// TIA Portal V16 export
// export: Created 2022-01-12T14:34:29.2729698Z, ExportSetting WithDefaults, DisplayName Totally Integrated Automation Portal, DisplayVersion V16 Update 4, DisplayName TIA Portal Version Control Interface, DisplayVersion V16 Update 2, DisplayName TIA Portal Openness, DisplayVersion V16 Update 4, DisplayName STEP 7 Professional, DisplayVersion V16 Update 4, DisplayName STEP 7 Safety, DisplayVersion V16, DisplayName WinCC Professional, DisplayVersion V16 Update 4
TYPE "typSygnałCiToObject"
// stored: IsFailsafeCompliant false
   STRUCT
      iCipLifeWord : UInt;   // lifeword:=lifeword+1 every 100ms
      iNrOfReqObjectToCip : UInt;   // Cip station tells you which object you want to clean
      iTimeToEndCip : UInt;   // remaining time to end of Cip process [seconds]
      bReqRouteToCip : Bool;   // Cip station request Object to set valves to Cip
      bCipIsActive : Bool;   // Cip statin informs of Active Cip process
      bReqPulloutTank : Bool;   // Cip station request Pullout process
      bReqStartReturnPump : Bool;   // Cip station request to start return pump (Cip-)
      bReqFlipValve : Bool;   // Cip station request Object ti flip valves
      bCipError : Bool;   // Cip station informs in Error
   END_STRUCT;
END_TYPE
